{attribute 'qualified_only'}
{attribute 'strict'}
TYPE ESeverity :
(
	none := 0,
	info := 1,
	warning := 2,
	error := 3
);
END_TYPE

(* stored: Version 1.1.0.1, ProductVersion 3.1.4024.9
   DUT ESeverity: Id {525d117c-6ba5-473d-b5d3-6507681629c0} *)
